(* PLC project Unnamed, Unknown Unnamed 1 *)
(* stored: creationDateTime 2024-03-18T04:34:39, modificationDateTime 2024-03-18T06:44:23 *)

PROGRAM program0
  VAR
    LocalVar0 AT %QW0.0.0.0 : UINT;
  END_VAR
  VAR
    LocalVar1 : UINT := 0;
  END_VAR

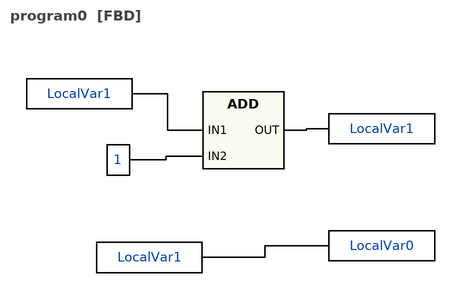
(* FBD diagram, written out as Structured Text *)
LocalVar1 := LocalVar1 + 1;
LocalVar0 := LocalVar1;
END_PROGRAM

CONFIGURATION config
  RESOURCE resource1 ON PLC
    TASK task0(INTERVAL := T#20ms, PRIORITY := 0);
    PROGRAM instance0 WITH task0 : program0;
  END_RESOURCE
END_CONFIGURATION
